// TIA Portal V16 export
// export: Created 2022-09-29T17:53:41.3528183Z, ExportSetting WithDefaults, DisplayName Totally Integrated Automation Portal, DisplayVersion V16, DisplayName TIA Portal Version Control Interface, DisplayVersion V16, DisplayName TIA Portal Openness, DisplayVersion V16, DisplayName STEP 7 Professional, DisplayVersion V16, DisplayName STEP 7 Safety, DisplayVersion V16, DisplayName WinCC Advanced, DisplayVersion V16
FUNCTION "Ciclo_Tratamento" : Void   // FC4, LAD
{ S7_Optimized_Access := 'TRUE' }
VERSION : 0.1
// stored: AutoNumber true, IsIECCheckEnabled false, SetENOAutomatically false, UDAEnableTagReadback false
   VAR_TEMP   // added for the SCL form of the ladder/FBD networks
      _w1 : Bool;
      _w2 : Bool;
   END_VAR
BEGIN

REGION Network 1: Etapa 1 (INÍCIO)
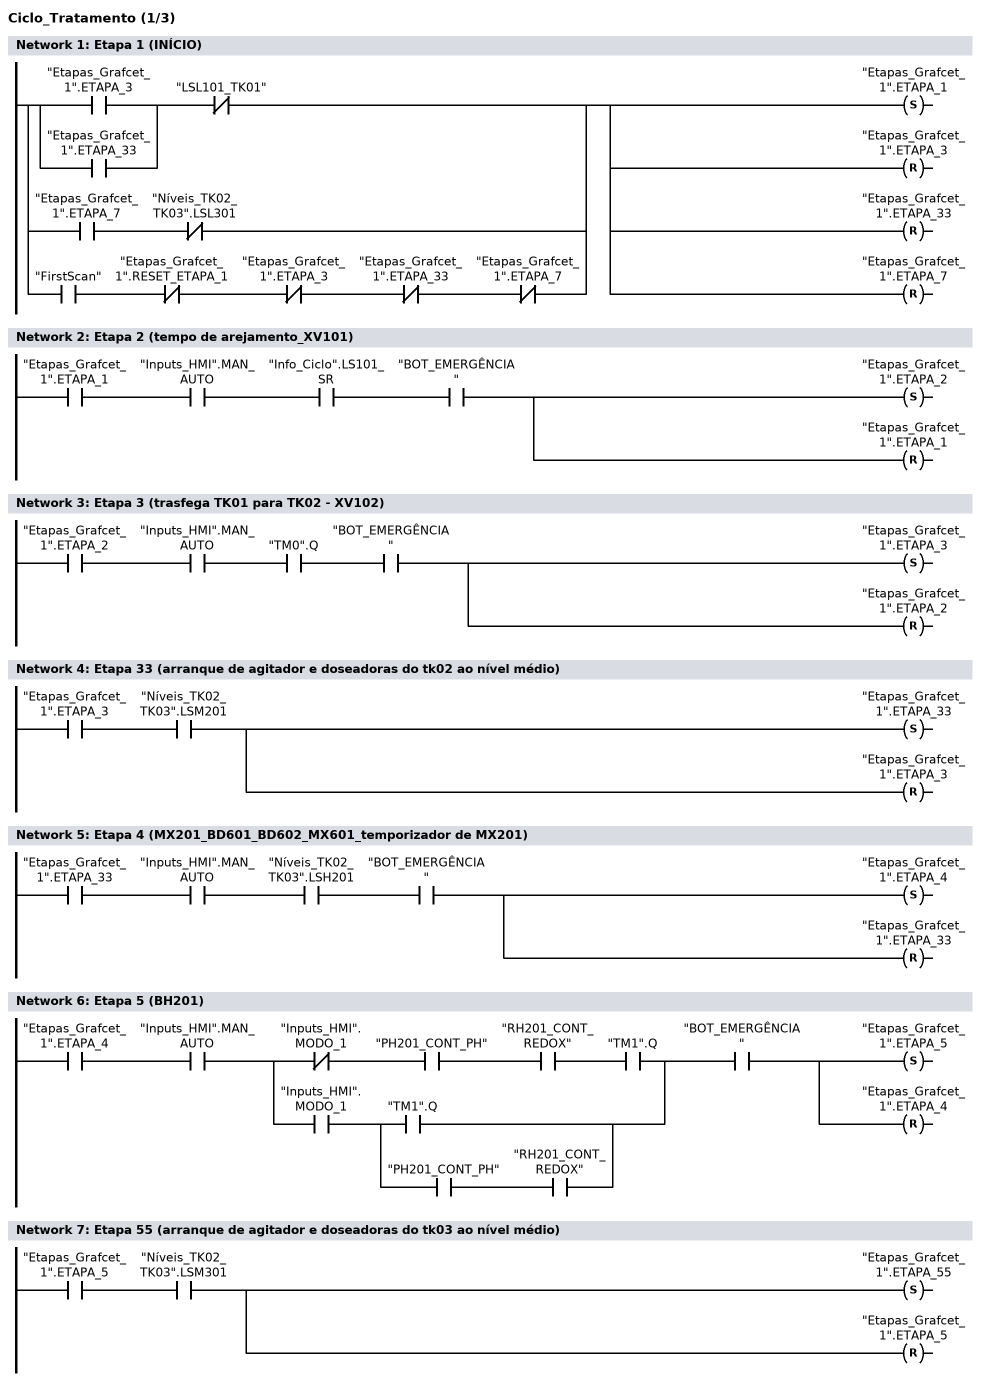
   RUNG wire#powerrail
      Contact( "Etapas_Grafcet_1".ETAPA_3 )
      wire#w1
      I_Contact( "LSL101_TK01" )
      wire#w2
      S_Coil( "Etapas_Grafcet_1".ETAPA_1 )
   END_RUNG
   RUNG wire#powerrail
      Contact( "Etapas_Grafcet_1".ETAPA_33 )
   END_RUNG wire#w1
   RUNG wire#powerrail
      Contact( "Etapas_Grafcet_1".ETAPA_7 )
      I_Contact( "Níveis_TK02_TK03".LSL301 )
   END_RUNG wire#w2
   RUNG wire#powerrail
      Contact( "FirstScan" )
      I_Contact( "Etapas_Grafcet_1".RESET_ETAPA_1 )
      I_Contact( "Etapas_Grafcet_1".ETAPA_3 )
      I_Contact( "Etapas_Grafcet_1".ETAPA_33 )
      I_Contact( "Etapas_Grafcet_1".ETAPA_7 )
   END_RUNG wire#w2
   RUNG wire#w2
      R_Coil( "Etapas_Grafcet_1".ETAPA_3 )
   END_RUNG
   RUNG wire#w2
      R_Coil( "Etapas_Grafcet_1".ETAPA_33 )
   END_RUNG
   RUNG wire#w2
      R_Coil( "Etapas_Grafcet_1".ETAPA_7 )
   END_RUNG
   // the same network as SCL:
   IF (("Etapas_Grafcet_1".ETAPA_3 OR "Etapas_Grafcet_1".ETAPA_33) AND NOT "LSL101_TK01") OR ("Etapas_Grafcet_1".ETAPA_7 AND NOT "Níveis_TK02_TK03".LSL301) OR ("FirstScan" AND NOT "Etapas_Grafcet_1".RESET_ETAPA_1 AND NOT "Etapas_Grafcet_1".ETAPA_3 AND NOT "Etapas_Grafcet_1".ETAPA_33 AND NOT "Etapas_Grafcet_1".ETAPA_7) THEN
       "Etapas_Grafcet_1".ETAPA_1 := TRUE;
   END_IF;
   #_w1 := (("Etapas_Grafcet_1".ETAPA_3 OR "Etapas_Grafcet_1".ETAPA_33) AND NOT "LSL101_TK01") OR ("Etapas_Grafcet_1".ETAPA_7 AND NOT "Níveis_TK02_TK03".LSL301) OR ("FirstScan" AND NOT "Etapas_Grafcet_1".RESET_ETAPA_1 AND NOT "Etapas_Grafcet_1".ETAPA_3 AND NOT "Etapas_Grafcet_1".ETAPA_33 AND NOT "Etapas_Grafcet_1".ETAPA_7);
   IF #_w1 THEN
       "Etapas_Grafcet_1".ETAPA_3 := FALSE;
       "Etapas_Grafcet_1".ETAPA_33 := FALSE;
       "Etapas_Grafcet_1".ETAPA_7 := FALSE;
   END_IF;
END_REGION

REGION Network 2: Etapa 2 (tempo de arejamento_XV101)
   RUNG wire#powerrail
      Contact( "Etapas_Grafcet_1".ETAPA_1 )
      Contact( "Inputs_HMI".MAN_AUTO )
      Contact( "Info_Ciclo".LS101_SR )
      Contact( "BOT_EMERGÊNCIA" )
      wire#w1
      S_Coil( "Etapas_Grafcet_1".ETAPA_2 )
   END_RUNG
   RUNG wire#w1
      R_Coil( "Etapas_Grafcet_1".ETAPA_1 )
   END_RUNG
   // the same network as SCL:
   IF "Etapas_Grafcet_1".ETAPA_1 AND "Inputs_HMI".MAN_AUTO AND "Info_Ciclo".LS101_SR AND "BOT_EMERGÊNCIA" THEN
       "Etapas_Grafcet_1".ETAPA_2 := TRUE;
       "Etapas_Grafcet_1".ETAPA_1 := FALSE;
   END_IF;
END_REGION

REGION Network 3: Etapa 3 (trasfega TK01 para TK02 - XV102)
   RUNG wire#powerrail
      Contact( "Etapas_Grafcet_1".ETAPA_2 )
      Contact( "Inputs_HMI".MAN_AUTO )
      Contact( "TM0".Q )
      Contact( "BOT_EMERGÊNCIA" )
      wire#w1
      S_Coil( "Etapas_Grafcet_1".ETAPA_3 )
   END_RUNG
   RUNG wire#w1
      R_Coil( "Etapas_Grafcet_1".ETAPA_2 )
   END_RUNG
   // the same network as SCL:
   IF "Etapas_Grafcet_1".ETAPA_2 AND "Inputs_HMI".MAN_AUTO AND "TM0".Q AND "BOT_EMERGÊNCIA" THEN
       "Etapas_Grafcet_1".ETAPA_3 := TRUE;
       "Etapas_Grafcet_1".ETAPA_2 := FALSE;
   END_IF;
END_REGION

REGION Network 4: Etapa 33 (arranque de agitador e doseadoras do tk02 ao nível médio)
   RUNG wire#powerrail
      Contact( "Etapas_Grafcet_1".ETAPA_3 )
      Contact( "Níveis_TK02_TK03".LSM201 )
      wire#w1
      S_Coil( "Etapas_Grafcet_1".ETAPA_33 )
   END_RUNG
   RUNG wire#w1
      R_Coil( "Etapas_Grafcet_1".ETAPA_3 )
   END_RUNG
   // the same network as SCL:
   IF "Etapas_Grafcet_1".ETAPA_3 AND "Níveis_TK02_TK03".LSM201 THEN
       "Etapas_Grafcet_1".ETAPA_33 := TRUE;
       "Etapas_Grafcet_1".ETAPA_3 := FALSE;
   END_IF;
END_REGION

REGION Network 5: Etapa 4 (MX201_BD601_BD602_MX601_temporizador de MX201)
   RUNG wire#powerrail
      Contact( "Etapas_Grafcet_1".ETAPA_33 )
      Contact( "Inputs_HMI".MAN_AUTO )
      Contact( "Níveis_TK02_TK03".LSH201 )
      Contact( "BOT_EMERGÊNCIA" )
      wire#w1
      S_Coil( "Etapas_Grafcet_1".ETAPA_4 )
   END_RUNG
   RUNG wire#w1
      R_Coil( "Etapas_Grafcet_1".ETAPA_33 )
   END_RUNG
   // the same network as SCL:
   IF "Etapas_Grafcet_1".ETAPA_33 AND "Inputs_HMI".MAN_AUTO AND "Níveis_TK02_TK03".LSH201 AND "BOT_EMERGÊNCIA" THEN
       "Etapas_Grafcet_1".ETAPA_4 := TRUE;
       "Etapas_Grafcet_1".ETAPA_33 := FALSE;
   END_IF;
END_REGION

REGION Network 6: Etapa 5 (BH201)
   RUNG wire#powerrail
      Contact( "Etapas_Grafcet_1".ETAPA_4 )
      Contact( "Inputs_HMI".MAN_AUTO )
      wire#w1
      I_Contact( "Inputs_HMI".MODO_1 )
      Contact( "PH201_CONT_PH" )
      Contact( "RH201_CONT_REDOX" )
      Contact( "TM1".Q )
      wire#w2
      Contact( "BOT_EMERGÊNCIA" )
      wire#w4
      S_Coil( "Etapas_Grafcet_1".ETAPA_5 )
   END_RUNG
   RUNG wire#w1
      Contact( "Inputs_HMI".MODO_1 )
      wire#w3
      Contact( "TM1".Q )
   END_RUNG wire#w2
   RUNG wire#w3
      Contact( "PH201_CONT_PH" )
      Contact( "RH201_CONT_REDOX" )
   END_RUNG wire#w2
   RUNG wire#w4
      R_Coil( "Etapas_Grafcet_1".ETAPA_4 )
   END_RUNG
   // the same network as SCL:
   IF "Etapas_Grafcet_1".ETAPA_4 AND "Inputs_HMI".MAN_AUTO AND ((NOT "Inputs_HMI".MODO_1 AND "PH201_CONT_PH" AND "RH201_CONT_REDOX" AND "TM1".Q) OR ("Inputs_HMI".MODO_1 AND ("TM1".Q OR ("PH201_CONT_PH" AND "RH201_CONT_REDOX")))) AND "BOT_EMERGÊNCIA" THEN
       "Etapas_Grafcet_1".ETAPA_5 := TRUE;
       "Etapas_Grafcet_1".ETAPA_4 := FALSE;
   END_IF;
END_REGION

REGION Network 7: Etapa 55 (arranque de agitador e doseadoras do tk03 ao nível médio)
   RUNG wire#powerrail
      Contact( "Etapas_Grafcet_1".ETAPA_5 )
      Contact( "Níveis_TK02_TK03".LSM301 )
      wire#w1
      S_Coil( "Etapas_Grafcet_1".ETAPA_55 )
   END_RUNG
   RUNG wire#w1
      R_Coil( "Etapas_Grafcet_1".ETAPA_5 )
   END_RUNG
   // the same network as SCL:
   IF "Etapas_Grafcet_1".ETAPA_5 AND "Níveis_TK02_TK03".LSM301 THEN
       "Etapas_Grafcet_1".ETAPA_55 := TRUE;
       "Etapas_Grafcet_1".ETAPA_5 := FALSE;
   END_IF;
END_REGION

REGION Network 8: Etapa 6 (MX301_BD603_BD604_MX603_MX604_temporizador de MX301)
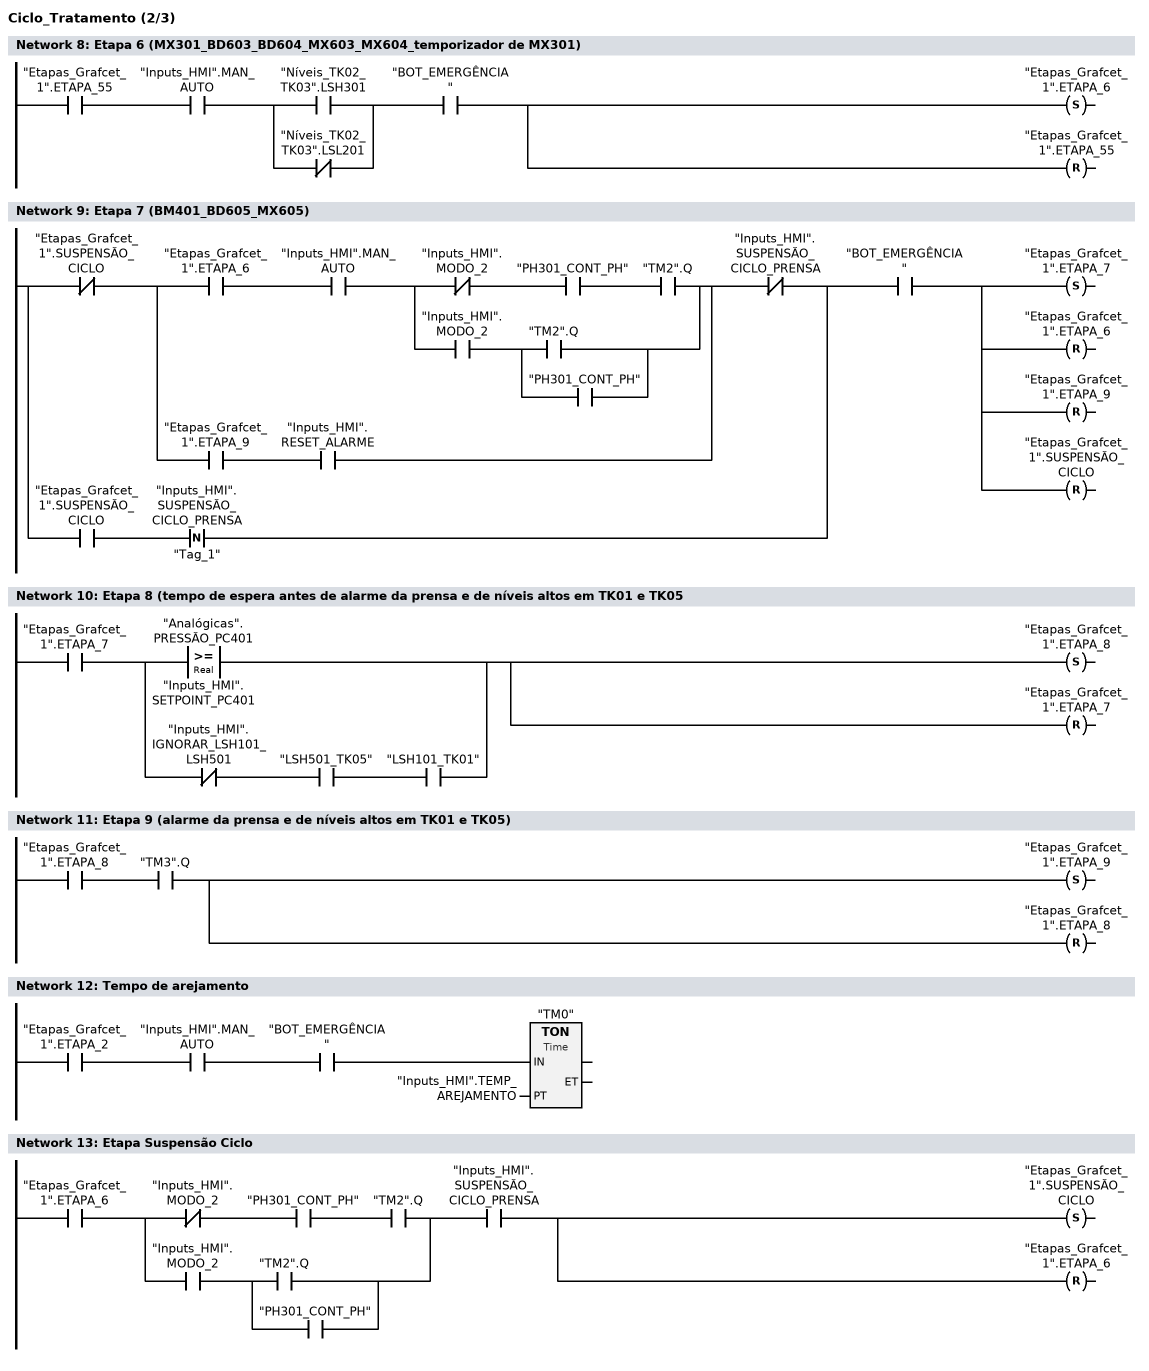
   RUNG wire#powerrail
      Contact( "Etapas_Grafcet_1".ETAPA_55 )
      Contact( "Inputs_HMI".MAN_AUTO )
      wire#w1
      Contact( "Níveis_TK02_TK03".LSH301 )
      wire#w2
      Contact( "BOT_EMERGÊNCIA" )
      wire#w3
      S_Coil( "Etapas_Grafcet_1".ETAPA_6 )
   END_RUNG
   RUNG wire#w1
      I_Contact( "Níveis_TK02_TK03".LSL201 )
   END_RUNG wire#w2
   RUNG wire#w3
      R_Coil( "Etapas_Grafcet_1".ETAPA_55 )
   END_RUNG
   // the same network as SCL:
   IF "Etapas_Grafcet_1".ETAPA_55 AND "Inputs_HMI".MAN_AUTO AND ("Níveis_TK02_TK03".LSH301 OR NOT "Níveis_TK02_TK03".LSL201) AND "BOT_EMERGÊNCIA" THEN
       "Etapas_Grafcet_1".ETAPA_6 := TRUE;
       "Etapas_Grafcet_1".ETAPA_55 := FALSE;
   END_IF;
END_REGION

REGION Network 9: Etapa 7 (BM401_BD605_MX605)
   RUNG wire#powerrail
      I_Contact( "Etapas_Grafcet_1".SUSPENSÃO_CICLO )
      wire#w1
      Contact( "Etapas_Grafcet_1".ETAPA_6 )
      Contact( "Inputs_HMI".MAN_AUTO )
      wire#w2
      I_Contact( "Inputs_HMI".MODO_2 )
      Contact( "PH301_CONT_PH" )
      Contact( "TM2".Q )
      wire#w3
      I_Contact( "Inputs_HMI".SUSPENSÃO_CICLO_PRENSA )
      wire#w5
      Contact( "BOT_EMERGÊNCIA" )
      wire#w6
      S_Coil( "Etapas_Grafcet_1".ETAPA_7 )
   END_RUNG
   RUNG wire#w2
      Contact( "Inputs_HMI".MODO_2 )
      wire#w4
      Contact( "TM2".Q )
   END_RUNG wire#w3
   RUNG wire#w4
      Contact( "PH301_CONT_PH" )
   END_RUNG wire#w3
   RUNG wire#w1
      Contact( "Etapas_Grafcet_1".ETAPA_9 )
      Contact( "Inputs_HMI".RESET_ALARME )
   END_RUNG wire#w3
   RUNG wire#powerrail
      Contact( "Etapas_Grafcet_1".SUSPENSÃO_CICLO )
      N_Contact(operand := "Inputs_HMI".SUSPENSÃO_CICLO_PRENSA, bit := "Tag_1")
   END_RUNG wire#w5
   RUNG wire#w6
      R_Coil( "Etapas_Grafcet_1".ETAPA_6 )
   END_RUNG
   RUNG wire#w6
      R_Coil( "Etapas_Grafcet_1".ETAPA_9 )
   END_RUNG
   RUNG wire#w6
      R_Coil( "Etapas_Grafcet_1".SUSPENSÃO_CICLO )
   END_RUNG
   // the same network as SCL:
   #_w1 := "Etapas_Grafcet_1".SUSPENSÃO_CICLO AND NOT "Inputs_HMI".SUSPENSÃO_CICLO_PRENSA AND "Tag_1";   // falling edge of "Inputs_HMI".SUSPENSÃO_CICLO_PRENSA
   "Tag_1" := "Inputs_HMI".SUSPENSÃO_CICLO_PRENSA;
   IF ((NOT "Etapas_Grafcet_1".SUSPENSÃO_CICLO AND (("Etapas_Grafcet_1".ETAPA_6 AND "Inputs_HMI".MAN_AUTO AND ((NOT "Inputs_HMI".MODO_2 AND "PH301_CONT_PH" AND "TM2".Q) OR ("Inputs_HMI".MODO_2 AND ("TM2".Q OR "PH301_CONT_PH")))) OR ("Etapas_Grafcet_1".ETAPA_9 AND "Inputs_HMI".RESET_ALARME)) AND NOT "Inputs_HMI".SUSPENSÃO_CICLO_PRENSA) OR #_w1) AND "BOT_EMERGÊNCIA" THEN
       "Etapas_Grafcet_1".ETAPA_7 := TRUE;
   END_IF;
   #_w2 := ((NOT "Etapas_Grafcet_1".SUSPENSÃO_CICLO AND (("Etapas_Grafcet_1".ETAPA_6 AND "Inputs_HMI".MAN_AUTO AND ((NOT "Inputs_HMI".MODO_2 AND "PH301_CONT_PH" AND "TM2".Q) OR ("Inputs_HMI".MODO_2 AND ("TM2".Q OR "PH301_CONT_PH")))) OR ("Etapas_Grafcet_1".ETAPA_9 AND "Inputs_HMI".RESET_ALARME)) AND NOT "Inputs_HMI".SUSPENSÃO_CICLO_PRENSA) OR #_w1) AND "BOT_EMERGÊNCIA";
   IF #_w2 THEN
       "Etapas_Grafcet_1".ETAPA_6 := FALSE;
       "Etapas_Grafcet_1".ETAPA_9 := FALSE;
       "Etapas_Grafcet_1".SUSPENSÃO_CICLO := FALSE;
   END_IF;
END_REGION

REGION Network 10: Etapa 8 (tempo de espera antes de alarme da prensa e de níveis altos em TK01 e TK05
   RUNG wire#powerrail
      Contact( "Etapas_Grafcet_1".ETAPA_7 )
      wire#w1
      { S7_Templates := "SrcType := Real" } GE_Contact(in1 := "Analógicas".PRESSÃO_PC401, in2 := "Inputs_HMI".SETPOINT_PC401)
      wire#w2
      S_Coil( "Etapas_Grafcet_1".ETAPA_8 )
   END_RUNG
   RUNG wire#w1
      I_Contact( "Inputs_HMI".IGNORAR_LSH101_LSH501 )
      Contact( "LSH501_TK05" )
      Contact( "LSH101_TK01" )
   END_RUNG wire#w2
   RUNG wire#w2
      R_Coil( "Etapas_Grafcet_1".ETAPA_7 )
   END_RUNG
   // the same network as SCL:
   IF "Etapas_Grafcet_1".ETAPA_7 AND (("Analógicas".PRESSÃO_PC401 >= "Inputs_HMI".SETPOINT_PC401) OR (NOT "Inputs_HMI".IGNORAR_LSH101_LSH501 AND "LSH501_TK05" AND "LSH101_TK01")) THEN
       "Etapas_Grafcet_1".ETAPA_8 := TRUE;
       "Etapas_Grafcet_1".ETAPA_7 := FALSE;
   END_IF;
END_REGION

REGION Network 11: Etapa 9 (alarme da prensa e de níveis altos em TK01 e TK05)
   RUNG wire#powerrail
      Contact( "Etapas_Grafcet_1".ETAPA_8 )
      Contact( "TM3".Q )
      wire#w1
      S_Coil( "Etapas_Grafcet_1".ETAPA_9 )
   END_RUNG
   RUNG wire#w1
      R_Coil( "Etapas_Grafcet_1".ETAPA_8 )
   END_RUNG
   // the same network as SCL:
   IF "Etapas_Grafcet_1".ETAPA_8 AND "TM3".Q THEN
       "Etapas_Grafcet_1".ETAPA_9 := TRUE;
       "Etapas_Grafcet_1".ETAPA_8 := FALSE;
   END_IF;
END_REGION

REGION Network 12: Tempo de arejamento
   RUNG wire#powerrail
      Contact( "Etapas_Grafcet_1".ETAPA_2 )
      Contact( "Inputs_HMI".MAN_AUTO )
      Contact( "BOT_EMERGÊNCIA" )
      { S7_Templates := "time_type := Time" } "TM0".TON(pt := "Inputs_HMI".TEMP_AREJAMENTO, et =>)
   END_RUNG
   // the same network as SCL:
   "TM0".TON(IN := "Etapas_Grafcet_1".ETAPA_2 AND "Inputs_HMI".MAN_AUTO AND "BOT_EMERGÊNCIA",
             PT := "Inputs_HMI".TEMP_AREJAMENTO);
END_REGION

REGION Network 13: Etapa Suspensão Ciclo
   RUNG wire#powerrail
      Contact( "Etapas_Grafcet_1".ETAPA_6 )
      wire#w1
      I_Contact( "Inputs_HMI".MODO_2 )
      Contact( "PH301_CONT_PH" )
      Contact( "TM2".Q )
      wire#w2
      Contact( "Inputs_HMI".SUSPENSÃO_CICLO_PRENSA )
      wire#w4
      S_Coil( "Etapas_Grafcet_1".SUSPENSÃO_CICLO )
   END_RUNG
   RUNG wire#w1
      Contact( "Inputs_HMI".MODO_2 )
      wire#w3
      Contact( "TM2".Q )
   END_RUNG wire#w2
   RUNG wire#w3
      Contact( "PH301_CONT_PH" )
   END_RUNG wire#w2
   RUNG wire#w4
      R_Coil( "Etapas_Grafcet_1".ETAPA_6 )
   END_RUNG
   // the same network as SCL:
   IF "Etapas_Grafcet_1".ETAPA_6 AND ((NOT "Inputs_HMI".MODO_2 AND "PH301_CONT_PH" AND "TM2".Q) OR ("Inputs_HMI".MODO_2 AND ("TM2".Q OR "PH301_CONT_PH"))) AND "Inputs_HMI".SUSPENSÃO_CICLO_PRENSA THEN
       "Etapas_Grafcet_1".SUSPENSÃO_CICLO := TRUE;
       "Etapas_Grafcet_1".ETAPA_6 := FALSE;
   END_IF;
END_REGION

REGION Network 14: Reset Suspensão Ciclo
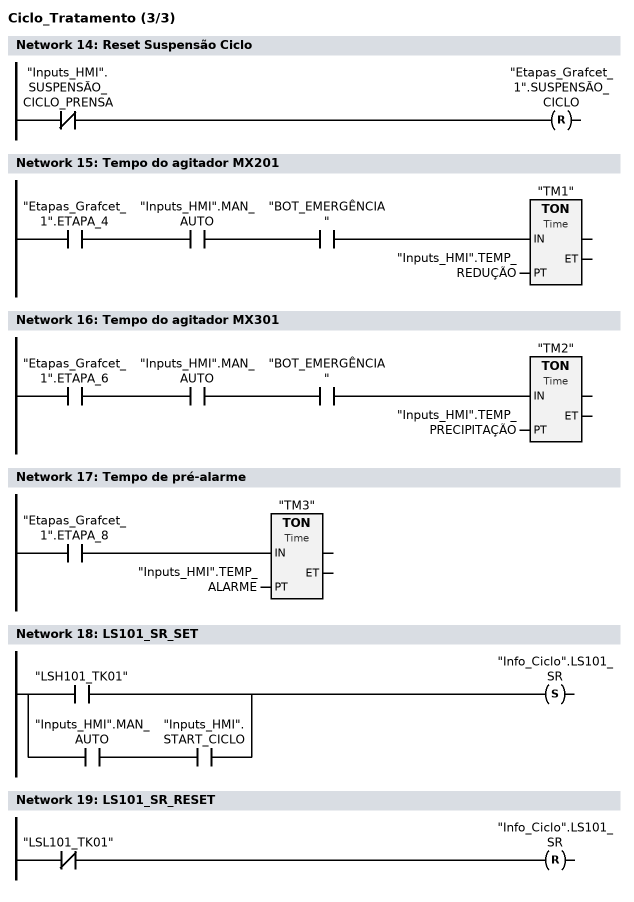
   RUNG wire#powerrail
      I_Contact( "Inputs_HMI".SUSPENSÃO_CICLO_PRENSA )
      R_Coil( "Etapas_Grafcet_1".SUSPENSÃO_CICLO )
   END_RUNG
   // the same network as SCL:
   IF NOT "Inputs_HMI".SUSPENSÃO_CICLO_PRENSA THEN "Etapas_Grafcet_1".SUSPENSÃO_CICLO := FALSE; END_IF;
END_REGION

REGION Network 15: Tempo do agitador MX201
   RUNG wire#powerrail
      Contact( "Etapas_Grafcet_1".ETAPA_4 )
      Contact( "Inputs_HMI".MAN_AUTO )
      Contact( "BOT_EMERGÊNCIA" )
      { S7_Templates := "time_type := Time" } "TM1".TON(pt := "Inputs_HMI".TEMP_REDUÇÃO, et =>)
   END_RUNG
   // the same network as SCL:
   "TM1".TON(IN := "Etapas_Grafcet_1".ETAPA_4 AND "Inputs_HMI".MAN_AUTO AND "BOT_EMERGÊNCIA",
             PT := "Inputs_HMI".TEMP_REDUÇÃO);
END_REGION

REGION Network 16: Tempo do agitador MX301
   RUNG wire#powerrail
      Contact( "Etapas_Grafcet_1".ETAPA_6 )
      Contact( "Inputs_HMI".MAN_AUTO )
      Contact( "BOT_EMERGÊNCIA" )
      { S7_Templates := "time_type := Time" } "TM2".TON(pt := "Inputs_HMI".TEMP_PRECIPITAÇÃO, et =>)
   END_RUNG
   // the same network as SCL:
   "TM2".TON(IN := "Etapas_Grafcet_1".ETAPA_6 AND "Inputs_HMI".MAN_AUTO AND "BOT_EMERGÊNCIA",
             PT := "Inputs_HMI".TEMP_PRECIPITAÇÃO);
END_REGION

REGION Network 17: Tempo de pré-alarme
   RUNG wire#powerrail
      Contact( "Etapas_Grafcet_1".ETAPA_8 )
      { S7_Templates := "time_type := Time" } "TM3".TON(pt := "Inputs_HMI".TEMP_ALARME, et =>)
   END_RUNG
   // the same network as SCL:
   "TM3".TON(IN := "Etapas_Grafcet_1".ETAPA_8, PT := "Inputs_HMI".TEMP_ALARME);
END_REGION

REGION Network 18: LS101_SR_SET
   RUNG wire#powerrail
      Contact( "LSH101_TK01" )
      wire#w1
      S_Coil( "Info_Ciclo".LS101_SR )
   END_RUNG
   RUNG wire#powerrail
      Contact( "Inputs_HMI".MAN_AUTO )
      Contact( "Inputs_HMI".START_CICLO )
   END_RUNG wire#w1
   // the same network as SCL:
   IF "LSH101_TK01" OR ("Inputs_HMI".MAN_AUTO AND "Inputs_HMI".START_CICLO) THEN
       "Info_Ciclo".LS101_SR := TRUE;
   END_IF;
END_REGION

REGION Network 19: LS101_SR_RESET
   RUNG wire#powerrail
      I_Contact( "LSL101_TK01" )
      R_Coil( "Info_Ciclo".LS101_SR )
   END_RUNG
   // the same network as SCL:
   IF NOT "LSL101_TK01" THEN "Info_Ciclo".LS101_SR := FALSE; END_IF;
END_REGION
END_FUNCTION
